// TIA Portal V21 export
DATA_BLOCK "JacketDrain"   // DB312
AUTHOR : PRECISE
FAMILY : PRECISE
// stored: AutoNumber false, InstanceOfName FB317, InstanceOfType FB
"FB317"
   // VAR_INPUT
   //    Enable : Bool;
   //    Disable : Bool;
   //    Fault : Bool;
   //    SecPulse : Bool;
   //    AlwaysTrue : Bool;
   //    StartConfirmationPopupSel : Bool;
   //    EndConfirmationPopupSel : Bool;
   //    SpargingModeSel : Int;
   //    SpargingTimebaseSel : Bool;
   //    SpargingLineSel : Bool;
   //    N2Sel : Int;
   //    SetDO : Real;
   //    SpargingTimeMin : Int;
   //    JdDelaySec : Int;
   //    PressuretoOpenVV : Real;
   //    PressuretoCloseVV : Real;
   //    ActualDO : Real;
   //    ActualPressure : Real;
   //    DelaytoOpenJd : Int;
   // END_VAR
   // VAR_OUTPUT
   //    PasValve : Bool;
   //    N2Valve : Bool;
   //    JdValve : Bool;
   //    JvValve : Bool;
   //    StartConfirmationPopup : Bool;
   //    EndConfirmationPopup : Bool;
   //    SpargingTimeMinPV : DInt;
   //    SpargingTimeSecPV : DInt;
   //    PrintTrigger : Bool;
   //    PrintWord : Int;
   //    PrintStatus : String[50];
   // END_VAR
   // VAR_IN_OUT
   //    Start : Bool;
   //    Stop : Bool;
   //    Close : Bool;
   //    StartConfirmationAck : Bool;
   //    EndConfirmationAck : Bool;
   //    SpareBtn1 : Bool;
   //    SpareBtn2 : Bool;
   //    SpareBtn3 : Bool;
   //    Running : Bool;
   //    Selected : Bool;
   //    Paused : Bool;
   //    StartConfirmationPopupTemp : Bool;
   //    EndConfirmationPopupTemp : Bool;
   //    SpargingStarted : Bool;
   //    SpargingOver : Bool;
   //    SpargingTimerRunning : Bool;
   // END_VAR
   // VAR
   //    ValveOnDelayPV : Int;
   //    ValveOffDelayPV : Int;
   //    PrintTriggerTemp : Bool;
   //    RE1 : Bool;
   //    RE2 : Bool;
   //    RE3 : Bool;
   //    RE4 : Bool;
   //    RE5 : Bool;
   //    RE6 : Bool;
   //    RE7 : Bool;
   //    SpargingTimer { S7_SetPoint := 'True'} : "FB101";
   //    PrintTriggerResetTimer { S7_SetPoint := 'True'} : TON_TIME;
   //    BtnResetTimer { S7_SetPoint := 'True'} : TON_TIME;
   // END_VAR
BEGIN
END_DATA_BLOCK
